{attribute 'linkalways'} 
{attribute 'no_explicit_call' := 'This FB is a CLASS and must be accessed using methods or properties'}
{attribute 'enable_dynamic_creation'}
FUNCTION_BLOCK Node_F_VN_GenerateColorMap EXTENDS Node
VAR
	ipColorMap : _ITcVnContainer;
    eColorMap : _ETcVnColorMap(ETcVnColorMap.TCVN_CM_AUTUMN);
    eColorMapSize : _ETcVnColorMapSize(ETcVnColorMapSize.TCVN_CMS_256);
    hrPrev : _HRESULT(S_OK);
	hresult : _HRESULT(S_OK);
END_VAR

METHOD PUBLIC  Clone : I_Node
VAR
	pNode : POINTER TO Node_F_VN_GenerateColorMap;
END_VAR
pNode := __NEW(Node_F_VN_GenerateColorMap);
Clone := pNode^;
END_METHOD

METHOD FB_init : BOOL
VAR_INPUT
	bInitRetains : BOOL; // if TRUE, the retain variables are initialized (warm start / cold start)
	bInCopyCode : BOOL;  // if TRUE, the instance afterwards gets moved into the copy code (online change)
END_VAR
AddInput('hrPrev', hrPrev);
AddOutput('ipColorMap', ipColorMap);
AddOutput('hresult',hresult);
AddParameter('eColorMap', eColorMap);
AddParameter('eColorMapSize', eColorMapSize);
END_METHOD

METHOD PROTECTED  OnExecute : HRESULT
hresult.Value := F_VN_GenerateColorMap(
	ipColorMap   := ipColorMap.Value,
	eColorMap := eColorMap.Value,
    eColorMapSize := eColorMapSize.Value, 
	hrPrev := hrPrev.Value);
END_METHOD

END_FUNCTION_BLOCK

(* stored: Version 1.1.0.1, ProductVersion 3.1.4024.13
   POU Node_F_VN_GenerateColorMap: Id {27e5698f-0f50-094d-35ab-3468fce1a159}, SpecialFunc None
   Folder Constructor: Id {e6188b16-79fe-0e80-079b-3a75fa65d5f3}
   Method Clone: Id {3503780f-73c0-0175-1345-5c43f2113088}
   Method FB_init: Id {8dddebcd-f373-0f5e-0f89-5e66023e0109}
   Method OnExecute: Id {7a45bbfe-3d8f-0629-14e9-194e60981cef} *)
